// Mitsubishi GX Works2 project: Tinh SUM   PLC: FX3U/FX3UC

PROGRAM MAIN
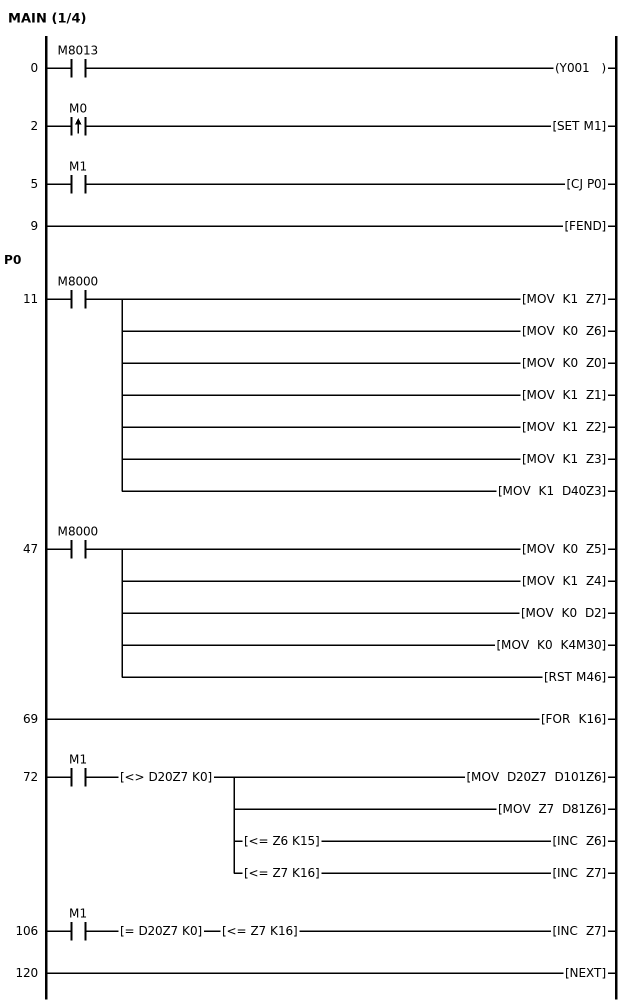
0     LD      M8013
      OUT     Y001
2     LDP     M0
      SET     M1
5     LD      M1
      CJ      P0
9     FEND
      P0
11    LD      M8000
      MOV     K1 Z7
      MOV     K0 Z6
      MOV     K0 Z0
      MOV     K1 Z1
      MOV     K1 Z2
      MOV     K1 Z3
      MOV     K1 D40Z3
47    LD      M8000
      MOV     K0 Z5
      MOV     K1 Z4
      MOV     K0 D2
      MOV     K0 K4M30
      RST     M46
69    FOR     K16
72    LD      M1
      AND<>   D20Z7 K0
      MOV     D20Z7 D101Z6
      MOV     Z7 D81Z6
      MPS
      AND<=   Z6 K15
      INC     Z6
      MPP
      AND<=   Z7 K16
      INC     Z7
106   LD      M1
      AND=    D20Z7 K0
      AND<=   Z7 K16
      INC     Z7
120   NEXT
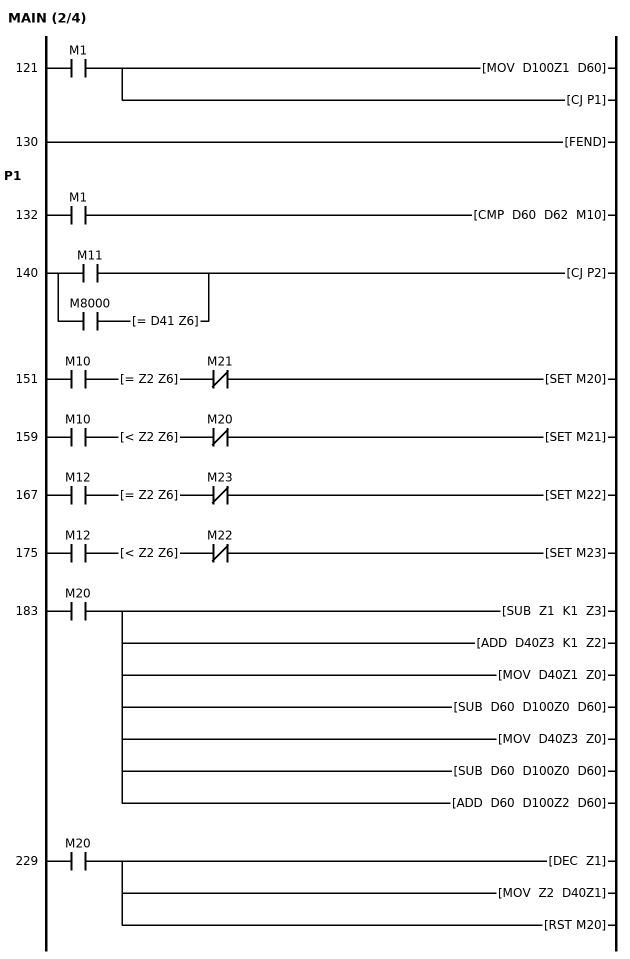
121   LD      M1
      MOV     D100Z1 D60
      CJ      P1
130   FEND
      P1
132   LD      M1
      CMP     D60 D62 M10
140   LD      M11
      LD      M8000
      AND=    D41 Z6
      ORB
      CJ      P2
151   LD      M10
      AND=    Z2 Z6
      ANI     M21
      SET     M20
159   LD      M10
      AND<    Z2 Z6
      ANI     M20
      SET     M21
167   LD      M12
      AND=    Z2 Z6
      ANI     M23
      SET     M22
175   LD      M12
      AND<    Z2 Z6
      ANI     M22
      SET     M23
183   LD      M20
      SUB     Z1 K1 Z3
      ADD     D40Z3 K1 Z2
      MOV     D40Z1 Z0
      SUB     D60 D100Z0 D60
      MOV     D40Z3 Z0
      SUB     D60 D100Z0 D60
      ADD     D60 D100Z2 D60
229   LD      M20
      DEC     Z1
      MOV     Z2 D40Z1
      RST     M20
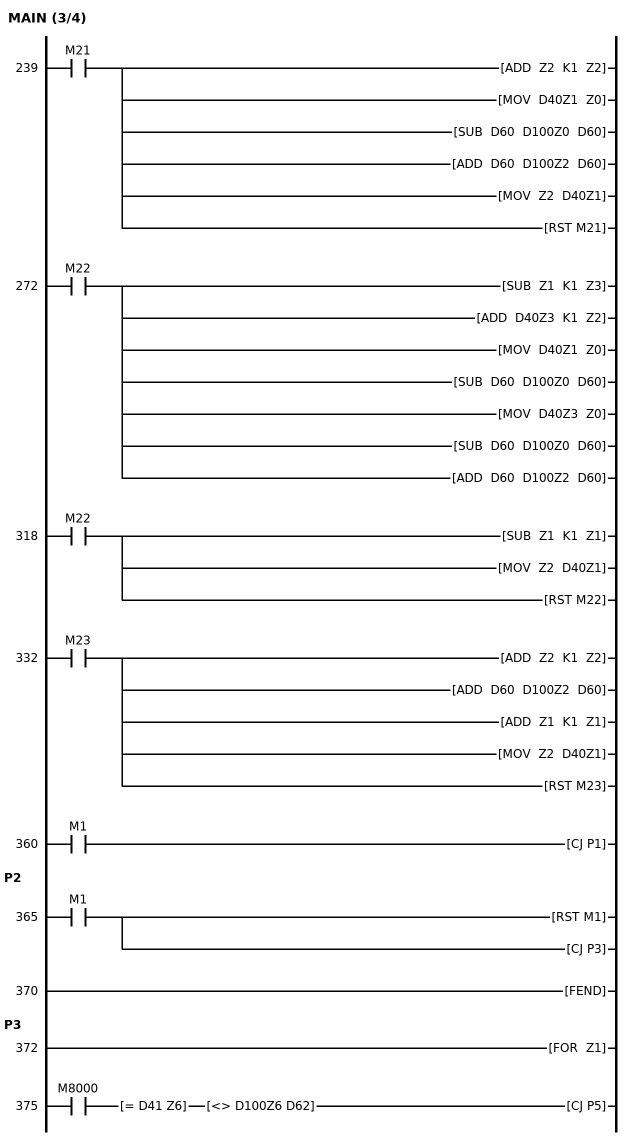
239   LD      M21
      ADD     Z2 K1 Z2
      MOV     D40Z1 Z0
      SUB     D60 D100Z0 D60
      ADD     D60 D100Z2 D60
      MOV     Z2 D40Z1
      RST     M21
272   LD      M22
      SUB     Z1 K1 Z3
      ADD     D40Z3 K1 Z2
      MOV     D40Z1 Z0
      SUB     D60 D100Z0 D60
      MOV     D40Z3 Z0
      SUB     D60 D100Z0 D60
      ADD     D60 D100Z2 D60
318   LD      M22
      SUB     Z1 K1 Z1
      MOV     Z2 D40Z1
      RST     M22
332   LD      M23
      ADD     Z2 K1 Z2
      ADD     D60 D100Z2 D60
      ADD     Z1 K1 Z1
      MOV     Z2 D40Z1
      RST     M23
360   LD      M1
      CJ      P1
      P2
365   LD      M1
      RST     M1
      CJ      P3
370   FEND
      P3
372   FOR     Z1
375   LD      M8000
      AND=    D41 Z6
      AND<>   D100Z6 D62
      CJ      P5
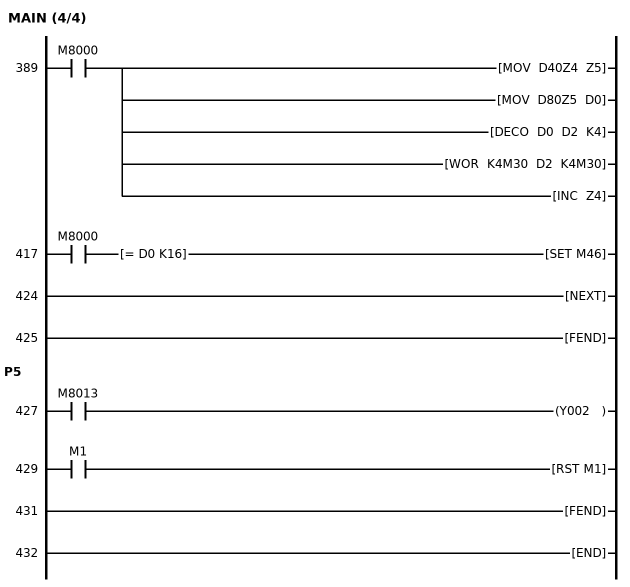
389   LD      M8000
      MOV     D40Z4 Z5
      MOV     D80Z5 D0
      DECO    D0 D2 K4
      WOR     K4M30 D2 K4M30
      INC     Z4
417   LD      M8000
      AND=    D0 K16
      SET     M46
424   NEXT
425   FEND
      P5
427   LD      M8013
      OUT     Y002
429   LD      M1
      RST     M1
431   FEND
432   END
END_PROGRAM
